FUNCTION p11_logicalFunction : BOOL
VAR_INPUT
	x1: BOOL;
	x2: BOOL;
END_VAR
VAR_OUTPUT
	y: BOOL;
END_VAR
VAR // added by the converter: edge detectors and wires of the graphical bodies
    _w1 : BOOL;
END_VAR

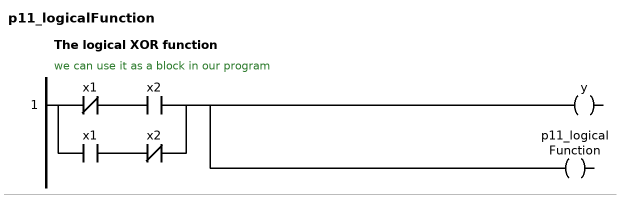
// NETWORK 1: The logical XOR function
// we can use it as a block in our program
_w1 := NOT x1 AND x2 OR x1 AND NOT x2;
y := _w1;
p11_logicalFunction := _w1;

END_FUNCTION

(* stored: Version 1.1.0.1, ProductVersion 3.1.4024.13
   POU p11_logicalFunction: Id {99c7539f-8c31-4abc-aeb1-62071c8d54a2}, SpecialFunc None *)
